(* IEC 61131-3 sources: com.logicals.lc3.webinar/usRTS_RPMControl_iSOC/src_FB_LIB_SAFE/Convert/UDINT, 5 files *)

(* ---- wTRUNC_UDINT_TO_UINT.iecst ---- *)
NAMESPACE logicals.web.standard
NAMESPACE convert

/*
 * Function block wrapper for IEC 61131-3 TO_UINT<br>
 * IN =  input value (UDINT)<br>
 * OUT = IN (UINT)<br>
 */
FUNCTION_BLOCK wTRUNC_UDINT_TO_UINT
	{ vNameAlignment:="center"; altName:="TRUNC_UDINT_TO_UINT"; bgColor:="Plum"; width:=180; hideIONames; }
	VAR_INPUT
		IN : UDINT;
	END_VAR
	VAR_OUTPUT
		OUT: UINT;
	END_VAR

	OUT := TO_UINT(IN:=IN, ENO=>ENO);
END_FUNCTION_BLOCK

END_NAMESPACE
END_NAMESPACE

(* ---- wTRUNC_UDINT_TO_USINT.iecst ---- *)
NAMESPACE logicals.web.standard
NAMESPACE convert

/*
 * Function block wrapper for IEC 61131-3 TO_USINT<br>
 * IN =  input value (UDINT)<br>
 * OUT = IN (USINT)<br>
 */
FUNCTION_BLOCK wTRUNC_UDINT_TO_USINT
	{ vNameAlignment:="center"; altName:="TRUNC_UDINT_TO_USINT"; bgColor:="Plum"; width:=180; hideIONames; }
	VAR_INPUT
		IN : UDINT;
	END_VAR
	VAR_OUTPUT
		OUT: USINT;
	END_VAR

	OUT := TO_USINT(IN:=IN, ENO=>ENO);
END_FUNCTION_BLOCK

END_NAMESPACE
END_NAMESPACE

(* ---- wUDINT_TO_DWORD.iecst ---- *)
NAMESPACE logicals.web.standard
NAMESPACE convert

/*
 * Function block wrapper for IEC 61131-3 TO_DWORD<br>
 * IN =  input value (UDINT)<br>
 * OUT = IN (DWORD)<br>
 */
FUNCTION_BLOCK wUDINT_TO_DWORD
	{ vNameAlignment:="center"; altName:="UDINT_TO_DWORD"; bgColor:="DodgerBlue"; width:=140; hideIONames; }
	VAR_INPUT
		IN : UDINT;
	END_VAR
	VAR_OUTPUT
		OUT: DWORD;
	END_VAR

	OUT := TO_DWORD(IN:=IN, ENO=>ENO);
END_FUNCTION_BLOCK

END_NAMESPACE
END_NAMESPACE

(* ---- wUDINT_TO_LINT.iecst ---- *)
NAMESPACE logicals.web.standard
NAMESPACE convert

/*
 * Function block wrapper for IEC 61131-3 TO_LINT<br>
 * IN =  input value (UDINT)<br>
 * OUT = IN (LINT)<br>
 */
FUNCTION_BLOCK wUDINT_TO_LINT
	{ vNameAlignment:="center"; altName:="UDINT_TO_LINT"; bgColor:="LightPink"; width:=140; hideIONames; }
	VAR_INPUT
		IN : UDINT;
	END_VAR
	VAR_OUTPUT
		OUT: LINT;
	END_VAR

	OUT := TO_LINT(IN:=IN, ENO=>ENO);
END_FUNCTION_BLOCK

END_NAMESPACE
END_NAMESPACE

(* ---- wUDINT_TO_ULINT.iecst ---- *)
NAMESPACE logicals.web.standard
NAMESPACE convert

/*
 * Function block wrapper for IEC 61131-3 TO_ULINT<br>
 * IN =  input value (UDINT)<br>
 * OUT = IN (ULINT)<br>
 */
FUNCTION_BLOCK wUDINT_TO_ULINT
	{ vNameAlignment:="center"; altName:="UDINT_TO_ULINT"; bgColor:="Plum"; width:=140; hideIONames; }
	VAR_INPUT
		IN : UDINT;
	END_VAR
	VAR_OUTPUT
		OUT: ULINT;
	END_VAR

	OUT := TO_ULINT(IN:=IN, ENO=>ENO);
END_FUNCTION_BLOCK

END_NAMESPACE
END_NAMESPACE
